FUNCTION_BLOCK GROUPING
  {SET_ATTRIBUTE(OpcUa, SERVICE)}
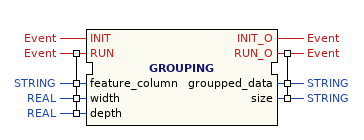
  EVENT_INPUT
    INIT;
    RUN WITH feature_column, width, depth; {SET_ATTRIBUTE(OpcUa, Method)}
  END_EVENT
  EVENT_OUTPUT
    INIT_O;
    RUN_O WITH groupped_data, size;
  END_EVENT
  VAR_INPUT
    feature_column : STRING; {SET_ATTRIBUTE(OpcUa, Variable)}
    width : REAL; {SET_ATTRIBUTE(OpcUa, Variable)}
    depth : REAL; {SET_ATTRIBUTE(OpcUa, Variable)}
  END_VAR
  VAR_OUTPUT
    groupped_data : STRING; {SET_ATTRIBUTE(OpcUa, Variable)}
    size : STRING; {SET_ATTRIBUTE(OpcUa, Variable)}
  END_VAR
END_FUNCTION_BLOCK
